INTERFACE ITF_ControlValve

PROPERTY EmergencyStatus : BOOL
GET
END_GET
END_PROPERTY

PROPERTY OperatingMode : BOOL
GET
END_GET
END_PROPERTY

PROPERTY OutputValue : REAL
GET
END_GET
END_PROPERTY

METHOD Reset : BOOL
VAR_INPUT
END_VAR
END_METHOD

METHOD SetMode : BOOL
VAR_INPUT
END_VAR
END_METHOD

METHOD SetValue : BOOL
VAR_INPUT
END_VAR
END_METHOD

END_INTERFACE

(* stored: Version 1.1.0.1, ProductVersion 3.1.4024.12
   Itf ITF_ControlValve: Id {ed7e0edb-f105-4663-98ee-2d269683d1ec}
   Folder Methods: Id {7ffb3e62-0840-4697-9d9c-5fdf97edce61}
   Folder Properties: Id {31babb0b-abf5-4aa4-a80f-1ed3ac86e8d7}
   Property EmergencyStatus: Id {b367e6dc-d1d7-440e-9012-0e6d604d9cfc}
   Get Get: Id {863f1d0c-cafa-47cc-b314-1734faaa5658}
   Property OperatingMode: Id {c9606c66-e346-4b53-8a78-5c7bfa43f6bc}
   Get Get: Id {03173b29-1607-4794-a1b3-9dce4479cf41}
   Property OutputValue: Id {19b61710-e94d-4c04-a43c-c44cef96f8a7}
   Get Get: Id {31deff39-c9ba-4d04-b188-cf975ce87f8c}
   Method Reset: Id {c3199e0c-0b11-4a5e-8fd6-5cdb75285f0d}
   Method SetMode: Id {5957c043-954f-40c1-99c5-6c5c6436ea64}
   Method SetValue: Id {50b712ca-ac5b-4e2b-82ac-09d1351b7c85} *)
